(* PLC project SafeLOGIC, BrAutomation SafeDESIGNER  5.24.1.0 *)
(* stored: companyURL http://www.br-automation.com, creationDateTime Sun Aug 10 20:37:49 2025 *)

PROGRAM ELAPSED_TIME

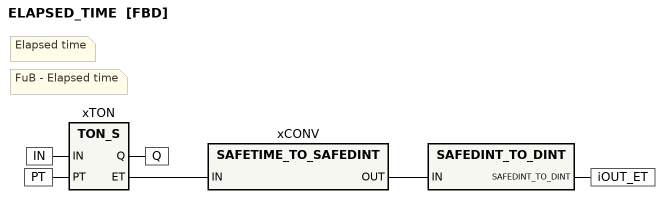
(* FBD diagram, written out as Structured Text *)
(* FuB - Elapsed time *)
(* Elapsed time *)
xTON(IN := IN, PT := PT);
Q := xTON.Q;
xCONV(IN := xTON.ET);
iOUT_ET := SAFEDINT_TO_DINT(xCONV.OUT);
END_PROGRAM
